TYPE TcaWorkpiecePlaceService :
STRUCT

END_STRUCT
END_TYPE

(* stored: Version 1.1.0.1
   DUT TcaWorkpiecePlaceService: Id {ded92dee-93a4-47f7-90ae-411824dbb7b3} *)
